// TIA Portal V17 export
// export: Created 2022-06-27T14:00:50.7140607Z, ExportSetting WithDefaults, DisplayName Totally Integrated Automation Portal, DisplayVersion V17 Update 3, DisplayName TIA Portal Openness, DisplayVersion V17 Update 3, DisplayName TIA Portal Version Control Interface, DisplayVersion V17, DisplayName SINAMICS Startdrive Advanced, DisplayVersion V17 Update1, DisplayName SINAMICS Startdrive G110M, G120, G120C, G120D, G120P, G115D, DisplayVersion V17 Update1, DisplayName SINAMICS Startdrive G130, G150, S120, S150, SINAMICS MV, S210, DisplayVersion V17 Update1, DisplayName STEP 7 Professional, DisplayVersion V17 Update 3, DisplayName STEP 7 Safety, DisplayVersion V17, DisplayName WinCC UA Professional, DisplayVersion V17 Update 3
VAR_GLOBAL   // PLC tag table "A6-1C"
   "F32-2C" AT %I0.0 : Bool;   // Proteção ventilador queimador
   "F33-4C" AT %I0.1 : Bool;   // Proteção válvula rotativa ciclone torrador
   "F33-6C" AT %I0.2 : Bool;   // Proteção bomba de aromatização torrador
   "F34-2C" AT %I0.3 : Bool;   // Proteção ventilador torrando
   "F34-4C" AT %I0.4 : Bool;   // Proteção ventilador secado
   "F34-6C" AT %I0.5 : Bool;   // Proteção ventilador esfriador
   "F35-2C" AT %I0.6 : Bool;   // Proteção eixo com pás câmara 1
   "F35-4C" AT %I0.7 : Bool;   // Proteção eixo com pás câmara 2
   "F36-2C" AT %I1.0 : Bool;   // Proteção insuflador ar ambiente câmara 1
   "F36-3C" AT %I1.1 : Bool;   // Proteção insuflador ar ambiente câmara 2
   "F36-5C" AT %I1.2 : Bool;   // Proteção válvula rotativa ciclone esfriador
   "F36-7C" AT %I1.3 : Bool;   // Proteção rosca sob esfriador
   "F36-8C" AT %I1.4 : Bool;   // Proteção rosca inclinada
   "F37-2C" AT %I1.5 : Bool;   // Proteção eixo com pás esfriador 1
   "F37-3C" AT %I1.6 : Bool;   // Proteção eixo com pás esfriador 2
   "F37-5C" AT %I1.7 : Bool;   // Proteção válvula rotativa ciclone 1 secador
   "F37-7C" AT %I2.0 : Bool;   // Proteção válvula rotativa ciclone 2 secador
   "F37-8C" AT %I2.1 : Bool;   // Proteção rosca sob ciclones
   "A56-2E_I2-2" AT %I2.2 : Bool;   // Reserva I2.2
   "U33-2D" AT %I2.3 : Bool;   // Ventilador queimador ligado
   "U35-2D" AT %I2.4 : Bool;   // Eixo com pás câmara 1 ligado
   "U35-4D" AT %I2.5 : Bool;   // Eixo com pás câmara 2 ligado
   "U37-2D" AT %I2.6 : Bool;   // Eixo com pás esfriador 1 ligado
   "U37-3D" AT %I2.7 : Bool;   // Eixo com pás esfriador 2 ligado
   "K98-4E" AT %I3.0 : Bool;   // Defeito queimador
   "K98-6E" AT %I3.1 : Bool;   // Queimador em funcionamento
   "K98-3E" AT %I3.2 : Bool;   // Ventilador queimador do combustor ligado
   "K43-2D" AT %I3.3 : Bool;   // Auxiliar falta de energia
   "KSV44-5C" AT %I3.4 : Bool;   // Relé de segurança ativado
   FCI AT %I3.5 : Bool;   // Fonte de componentes internos OK
   FCE AT %I3.6 : Bool;   // Fonte de componentes externos OK
   "A56-2E_I3-7" AT %I3.7 : Bool;   // Reserva I3.7
   "KSV46-4C" AT %I4.0 : Bool;   // Relé de segurança câmara 1 acionado
   "KSV46-8C" AT %I4.1 : Bool;   // Relé de segurança câmara 2 acionado
   "KSV47-4C" AT %I4.2 : Bool;   // Relé de segurança esfriador 1 acionado
   "KSV47-8C" AT %I4.3 : Bool;   // Relé de segurança esfriador 2 acionado
   "A58-2E_I4-4" AT %I4.4 : Bool;   // Reserva I4.4
   "A58-2E_I4-5" AT %I4.5 : Bool;   // Reserva I4.5
   "A58-2E_I4-6" AT %I4.6 : Bool;   // Reserva I4.6
   "A58-2E_I4-7" AT %I4.7 : Bool;   // Reserva I4.7
   "S59-2C" AT %I5.0 : Bool;   // Botão emergência água câmara 1 acionado
   "S59-3C" AT %I5.1 : Bool;   // Botão emergência água esfriador 1 acionado
   "S59-4C" AT %I5.2 : Bool;   // Botão emergência água câmara 2 acionado
   "S59-5C" AT %I5.3 : Bool;   // Botão emergência água esfriador 2 acionado
   "S59-6C" AT %I5.4 : Bool;   // Botão desliga combustor acionado
   TCTL AT %I5.5 : Bool;   // Transporte de café torrado ligado
   "A58-2E_I5-6" AT %I5.6 : Bool;   // Reserva I5.6
   "A58-2E_I5-7" AT %I5.7 : Bool;   // Reserva I5.7
   "ZSV46-2C" AT %I6.0 : Bool;   // Fim de cruso de segurança acionamento manual câmara 1
   "ZSV46-6C" AT %I6.1 : Bool;   // Fim de cruso de segurança acionamento manual câmara 2
   "ZSV47-2C" AT %I6.2 : Bool;   // Fim de cruso de segurança acionamento manual esfriador 1
   "ZSV47-6C" AT %I6.3 : Bool;   // Fim de cruso de segurança acionamento manual esfriador 2
   "G43-4C-1" AT %I6.4 : Bool;   // Nobreak status bateria baixa
   "G43-4C-2" AT %I6.5 : Bool;   // Nobreak status de rede
   "A60-2E_I6-6" AT %I6.6 : Bool;   // Reserva I6.6
   "A60-2E_I6-7" AT %I6.7 : Bool;   // Reserva I6.7
   "A60-2E_I7-0" AT %I7.0 : Bool;   // Reserva I7.0
   "A60-2E_I7-1" AT %I7.1 : Bool;   // Reserva I7.1
   "A60-2E_I7-2" AT %I7.2 : Bool;   // Reserva I7.2
   "A60-2E_I7-3" AT %I7.3 : Bool;   // Reserva I7.3
   "A60-2E_I7-4" AT %I7.4 : Bool;   // Reserva I7.4
   "A60-2E_I7-5" AT %I7.5 : Bool;   // Reserva I7.5
   "A60-2E_I7-6" AT %I7.6 : Bool;   // Reserva I7.6
   "A60-2E_I7-7" AT %I7.7 : Bool;   // Reserva I7.7
   "K62-2E" AT %Q0.0 : Bool;   // Auxiliar acionamento ventilador combustor
   "KM62-3E" AT %Q0.1 : Bool;   // Válvula rotativa ciclone torrador
   "K62-4E" AT %Q0.2 : Bool;   // Auxiliar bomba de aromatização
   "K62-5E" AT %Q0.3 : Bool;   // Auxiliar acionamento eixo com pás câmara 1
   "K62-6E" AT %Q0.4 : Bool;   // Auxiliar acionamento eixo com pás câmara 2
   "KM62-7E" AT %Q0.5 : Bool;   // Válvula rotattiva ciclone esfriador
   "KM62-8E" AT %Q0.6 : Bool;   // Rosca sob esfriadores
   "KM62-9E" AT %Q0.7 : Bool;   // Rosca inclinada
   "K63-2E" AT %Q1.0 : Bool;   // Auxiliar acionamento eixo com pás esfriador 1
   "K63-3E" AT %Q1.1 : Bool;   // Auxiliar acionamento eixo com pás esfriador 2
   "KM63-4E" AT %Q1.2 : Bool;   // Válvula rotativa ciclone 1 secador
   "KM63-5E" AT %Q1.3 : Bool;   // Válvula rotativa ciclone 2 secador
   "KM63-6E" AT %Q1.4 : Bool;   // Rosca sob ciclones
   "K63-7E" AT %Q1.5 : Bool;   // Sinal pedido de café cru silo 1
   "K63-8E" AT %Q1.6 : Bool;   // Sinal pedido de café cru silo 2
   "A62-2E_Q1-7" AT %Q1.7 : Bool;   // Reserva Q1.7
   "K64-2E" AT %Q2.0 : Bool;   // Pedido para ligar trasnporte café torrado via catador
   "K64-3E" AT %Q2.1 : Bool;   // Pedido para ligar trasnporte café torrado via HVH
   "K64-4E" AT %Q2.2 : Bool;   // Auxiliar reset combustor
   "K64-5E" AT %Q2.3 : Bool;   // Auxiliar liga combustor
   "K64-6E" AT %Q2.4 : Bool;   // Seleção de combustível combustor
   "A64-2E_Q2-5" AT %Q2.5 : Bool;   // Reserva Q2.5
   "A64-2E_Q2-6" AT %Q2.6 : Bool;   // Reserva Q2.6
   "A64-2E_Q2-7" AT %Q2.7 : Bool;   // Reserva Q2.7
   "K65-2A" AT %Q3.0 : Bool;   // Auxiliar energiza programador de chama combustor
   "H65-3D-VE" AT %Q3.1 : Bool;   // Lâmpada sistema normal
   "H65-3D-VO" AT %Q3.2 : Bool;   // Lâmpada sistema em alarme
   "H65-3D-AS" AT %Q3.3 : Bool;   // Alarme sonoro
   "A64-2E_Q3-4" AT %Q3.4 : Bool;   // Alarme sonoro
   "A64-2E_Q3-5" AT %Q3.5 : Bool;   // Reserva Q3.5
   "A64-2E_Q3-6" AT %Q3.6 : Bool;   // Reserva Q3.6
   "A64-2E_Q3-7" AT %Q3.7 : Bool;   // Reserva Q3.7
   EnergyMeterUnkown AT %IW116 : Int;
   "Apparent power L1" AT %IW118 : Int;
   "Apparent power L1(1)" AT %IW120 : Int;
   "Apparent power L2" AT %IW122 : Int;
   "Apparent power L2(1)" AT %IW124 : Int;
   "Apparent power L3" AT %IW126 : Int;
   "Apparent power L3(1)" AT %IW128 : Int;
   "Total apparent power L1L2L3" AT %IW130 : Int;
   "Total apparent power L1L2L3(1)" AT %IW132 : Int;
   "Active power L1" AT %IW134 : Int;
   "Active power L1(1)" AT %IW136 : Int;
   "Active power L2" AT %IW138 : Int;
   "Active power L2(1)" AT %IW140 : Int;
   "Active power L3" AT %IW142 : Int;
   "Active power L3(1)" AT %IW144 : Int;
   "Total active power L1L2L3" AT %IW146 : Int;
   "Total active power L1L2L3(1)" AT %IW148 : Int;
   "Reactive power L1" AT %IW150 : Int;
   "Reactive power L1(1)" AT %IW152 : Int;
   "Reactive power L2" AT %IW154 : Int;
   "Reactive power L2(1)" AT %IW156 : Int;
   "Reactive power L3" AT %IW158 : Int;
   "Reactive power L3(1)" AT %IW160 : Int;
   "Total reactive power L1L2L3" AT %IW162 : Int;
   "Total reactive power L1L2L3(1)" AT %IW164 : Int;
   "Total apparent energy L1L2L3" AT %IW166 : Int;
   "Total apparent energy L1L2L3(1)" AT %IW168 : Int;
   "Total active energy L1L2L3" AT %IW170 : Int;
   "Total active energy L1L2L3(1)" AT %IW172 : Int;
   "Total reactive energy L1L2L3" AT %IW174 : Int;
   "Total reactive energy L1L2L3(1)" AT %IW176 : Int;
   "Current L1" AT %IW178 : Int;
   "Current L1(1)" AT %IW180 : Int;
   "Current L2" AT %IW182 : Int;
   "Current L2(1)" AT %IW184 : Int;
   "Current L3" AT %IW186 : Int;
   "Current L3(1)" AT %IW188 : Int;
END_VAR
